TYPE AxesTargetStatuses :
STRUCT
	healthStatus: HealthStatus;
END_STRUCT
END_TYPE

(* stored: Version 1.1.0.1, ProductVersion 3.1.4019.2
   DUT AxesTargetStatuses: Id {4d580295-6719-4b28-a90d-8e7987cca57d} *)
